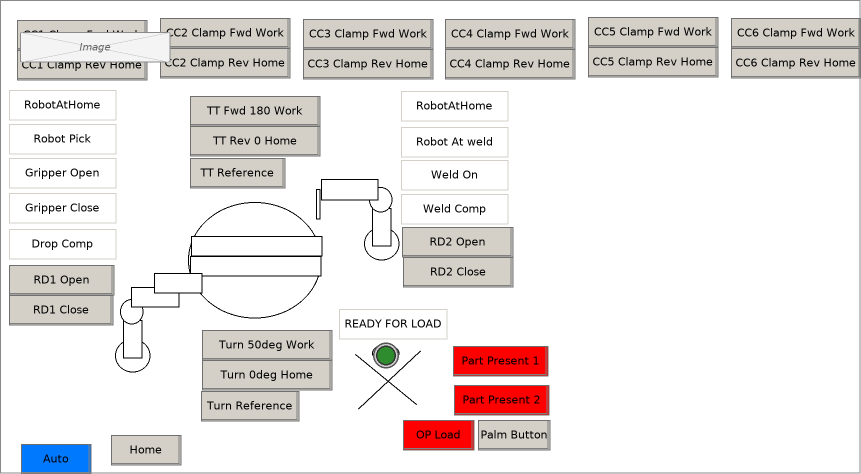
VISUALIZATION Clamp  // 861x474
    Button (17,20 130x30), "CC1 Clamp Fwd Work", colour toggle: IO.FixtureOutput.o_CC1_CLAMPING_UNIT1_3_WP
        tap HMI.CC1_Clamp_FwdCmd
    Button (17,50 130x30), "CC1 Clamp Rev Home", colour toggle: IO.FixtureOutput.o_CC1_CLAMPING_UNIT1_3_HP
        tap HMI.CC1_Clamp_RevCmd
    Button (160,18 130x30), "CC2 Clamp Fwd Work", colour toggle: IO.FixtureOutput.o_CC2_CLAMPING_UNIT2_3_WP
        tap HMI.CC2_Clamp_FwdCmd
    Button (160,48 130x30), "CC2 Clamp Rev Home", colour toggle: IO.FixtureOutput.o_CC2_CLAMPING_UNIT2_3_HP
        tap HMI.CC2_Clamp_RevCmd
    Button (303,19 130x30), "CC3 Clamp Fwd Work", colour toggle: IO.FixtureOutput.o_CC3_CLAMPING_UNIT3_3_WP
        tap HMI.CC3_Clamp_FwdCmd
    Button (303,49 130x30), "CC3 Clamp Rev Home", colour toggle: IO.FixtureOutput.o_CC3_CLAMPING_UNIT3_3_HP
        tap HMI.CC3_Clamp_RevCmd
    Button (445,19 130x30), "CC4 Clamp Fwd Work", colour toggle: IO.FixtureOutput.o_CC4_CLAMPING_UNIT4_3_WP
        tap HMI.CC4_Clamp_FwdCmd
    Button (445,49 130x30), "CC4 Clamp Rev Home", colour toggle: IO.FixtureOutput.o_CC4_CLAMPING_UNIT4_3_HP
        tap HMI.CC4_Clamp_RevCmd
    Button (588,17 130x30), "CC5 Clamp Fwd Work", colour toggle: IO.FixtureOutput.o_CC5_CLAMPING_UNIT5_1_WP
        tap HMI.CC5_Clamp_FwdCmd
    Button (588,47 130x30), "CC5 Clamp Rev Home", colour toggle: IO.FixtureOutput.o_CC5_CLAMPING_UNIT5_1_HP
        tap HMI.CC5_Clamp_RevCmd
    Button (731,18 130x30), "CC6 Clamp Fwd Work", colour toggle: IO.FixtureOutput.o_CC6_CLAMPING_UNIT6_1_WP
        tap HMI.CC6_Clamp_FwdCmd
    Button (731,48 130x30), "CC6 Clamp Rev Home", colour toggle: IO.FixtureOutput.o_CC6_CLAMPING_UNIT6_1_HP
        tap HMI.CC6_Clamp_RevCmd
    Button (9,265 105x30), "RD1 Open", colour toggle: IO.RD1.i_RD_Sensor_Open
        tap HMI.RD1_OpenCmd
    Button (9,295 104x30), "RD1 Close", colour toggle: IO.RD1.i_RD_Sensor_Close
        tap HMI.RD1_CloseCmd
    Button (402,227 111x30), "RD2 Open", colour toggle: IO.RD2.i_RD_Sensor_Open
        tap HMI.RD2_OpenCmd
    Button (403,257 110x30), "RD2 Close", colour toggle: IO.RD2.i_RD_Sensor_Close
        tap HMI.RD2_CloseCmd
    Button (190,96 130x30), "TT Fwd 180 Work", colour toggle: IO.TurnTableOutput.o_TurnTable_FWD_SENSOR
        tap HMI.TurnTableFwdCmd
    Button (190,126 130x30), "TT Rev 0 Home", colour toggle: IO.TurnTableOutput.o_TurnTable_REV_SENSOR
        tap HMI.TurnTableRevCmd
    Button (190,158 95x30), "TT Reference", colour toggle: IO.TurnTableOutput.o_TurnTable_REF_SENSOR
        tap HMI.TurnTableRef
    Ellipse (188,202 133x116)
    Button (202,330 130x30), "Turn 50deg Work", colour toggle: IO.Turn.o_Turn_FWD_SENSOR
        tap HMI.TurnFwdCmd
    Button (202,360 130x30), "Turn 0deg Home", colour toggle: IO.Turn.o_Turn_REV_SENSOR
        tap HMI.TurnRevCmd
    Button (201,391 98x30), "Turn Reference", colour toggle: IO.Turn.o_Turn_REF_SENSOR
        tap HMI.TurnRef
    Rectangle (190,256 131x20), colour toggle: Memory.Stat_Parts_Lvl2_Present
    Ellipse (372,344 27x18)
    Line (355,354) (416,404)
    Line (420,351) (358,409)
    Image (20,32 150x30)
    Button (403,420 71x30), "OP Load", colour toggle: Memory.In_Operator_Outside_Cell
        toggle Memory.In_Operator_Outside_Cell
    Button (453,346 95x30), "Part Present 1", colour toggle: Memory.Stat_Parts_Lvl1_Present
        toggle Memory.Stat_Parts_Lvl1_Present
    Button (454,385 95x30), "Part Present 2", colour toggle: Memory.Stat_Parts_Lvl2_Present
        toggle Memory.Stat_Parts_Lvl2_Present
    Button (478,420 72x30), "Palm Button", colour toggle: Memory.In_PalmButton_Pushed
        tap Memory.In_PalmButton_Pushed
    Button (21,444 70x30), "Auto", colour toggle: Memory.AutoMode
        toggle Memory.AutoMode
    Button (111,435 70x30), "Home", colour toggle: HMI.Home
        tap HMI.Home
    Ellipse (115,339 35x33)
    Rectangle (123,320 19x38)
    Ellipse (120,299 23x25)
    Rectangle (131,287 48x20), angle 331
    Rectangle (154,273 48x20), angle 236, colour toggle: RobotInterface.HDL_HandlingToCell.Gripper1ClosedAck
    Ellipse (364,227 35x33)
    Rectangle (372,208 19x38)
    Ellipse (369,187 23x25)
    Rectangle (321,179 57x21), angle 13
    Rectangle (316,189 4x30), angle 17, colour toggle: WeldRobotInterface.TorchOn
    Lamp1 (371,338 30x35), variable: HMI.ReadyForLoad, style: Lamp-Lamp1-Green
    Textfield (339,309 108x30), "READY FOR LOAD"
    Textfield (9,90 107x30), "RobotAtHome", text variable: RobotInterface.RobotAtHome, colour toggle: RobotInterface.RobotAtHome
    Textfield (9,124 107x30), "Robot Pick", text variable: RobotInterface.HDL_HandlingToCell.PickJobProceed, colour toggle: RobotInterface.HDL_HandlingToCell.PickJobProceed
    Textfield (9,158 107x30), "Gripper Open", text variable: RobotInterface.HDL_HandlingToCell.Gripper1OpenedAck, colour toggle: RobotInterface.HDL_HandlingToCell.Gripper1OpenedAck
    Textfield (9,193 107x30), "Gripper Close", text variable: RobotInterface.HDL_HandlingToCell.Gripper1ClosedAck, colour toggle: RobotInterface.HDL_HandlingToCell.Gripper1ClosedAck
    Textfield (9,229 107x30), "Drop Comp", text variable: RobotInterface.HDL_HandlingToCell.DropJobProceed, colour toggle: RobotInterface.HDL_HandlingToCell.PickJobOK
    Textfield (401,91 107x30), "RobotAtHome", text variable: WeldRobotInterface.RobotAtHome, colour toggle: WeldRobotInterface.RobotAtHome
    Textfield (401,160 107x30), "Weld On", text variable: WeldRobotInterface.TorchOn, colour toggle: WeldRobotInterface.TorchOn
    Textfield (401,127 107x30), "Robot At weld", text variable: WeldRobotInterface.RobotAtWeldPosition, colour toggle: WeldRobotInterface.RobotAtWeldPosition
    Textfield (401,194 107x30), "Weld Comp", text variable: Memory.In_Welding_Cycle_Complete, colour toggle: Memory.In_Welding_Cycle_Complete
    Rectangle (191,236 131x20), colour toggle: Memory.Stat_Parts_Lvl1_Present
END_VISUALIZATION

(* stored: Version 1.1.0.1, ProductVersion 3.1.4024.16
   Visu Clamp: Id {0ac5aced-59f8-4969-9650-e885bc783351} *)
